// TIA Portal V19 export
TYPE "udt_FComm"
// stored: Access Published, IsFailsafeCompliant true
   STRUCT
      EstopLocal : Bool;   // Emergency stop that stops only near devices
      EstopGlobal : Bool;   // Emergency stop that stops all devices
      Door_Ok : Bool;   // Cumulative of door OK
      Door_NormalStop : Bool;   // Cumulative of door normal stops
      Door_SafeStop : Bool;   // Cumulative of door safe stops
      _05 : Bool;
      LightCurtain_Ok : Bool;   // Input of lgiht curtain that divide 2 plcs
      _07 : Bool;
      _08 : Bool;
      EntryEnable : Bool;   // Door entry enable
      _10 : Bool;
      _11 : Bool;
      _12 : Bool;
      _13 : Bool;
      _14 : Bool;
      CommOk : Bool;   // 1=OK
   END_STRUCT;
END_TYPE
